FUNCTION_BLOCK FB_LedOff
VAR_INPUT
END_VAR
VAR_OUTPUT
END_VAR
VAR
	state : INT := 0;
	fbSerialSend : FB_SerialCom;
	d0 : BYTE := 16#01;
	d1 : BYTE := 16#44;
	d2 : BYTE := 16#00;
	d3 : BYTE := 16#13;
	d4 : BYTE := 16#00;
	fbSendData : SendData;
END_VAR

(*
BackGroundEL.stOut_EL6002_MB.D[0] := 16#01;
BackGroundEL.stOut_EL6002_MB.D[1] := 16#44;
BackGroundEL.stOut_EL6002_MB.D[2] := 16#00;
BackGroundEL.stOut_EL6002_MB.D[3] := 16#13;
BackGroundEL.stOut_EL6002_MB.D[4] := 16#00;
*)
(*
CASE state OF 
0:
fbSerialSend(
	TxBuffer := GVL.TxBufferEL_MB,
	RxBuffer := GVL.RxBufferEL_MB,
	fbSendData := fbSendData.pSendData,
	Busy =>,
	Error =>
	);
	IF fbSerialSend.Busy = FALSE THEN
		state := state + 1;
	END_IF
1:
fbSerialSend(
	TxBuffer := GVL.TxBufferEL_MB,
	RxBuffer := GVL.RxBufferEL_MB,
	fbSendData := d0,
	Busy =>,
	Error =>
	);
	IF fbSerialSend.Busy = FALSE THEN
		state := state + 1;
	END_IF
2:
fbSerialSend(
	TxBuffer := GVL.TxBufferEL_MB,
	RxBuffer := GVL.RxBufferEL_MB,
	fbSendData := d0,
	Busy =>,
	Error =>
	);
	IF fbSerialSend.Busy = FALSE THEN
		state := state + 1;
	END_IF
3:
fbSerialSend(
	TxBuffer := GVL.TxBufferEL_MB,
	RxBuffer := GVL.RxBufferEL_MB,
	fbSendData := d0,
	Busy =>,
	Error =>
	);
	IF fbSerialSend.Busy = FALSE THEN
		state := state + 1;
	END_IF
4:
fbSerialSend(
	TxBuffer := GVL.TxBufferEL_MB,
	RxBuffer := GVL.RxBufferEL_MB,
	fbSendData := d0,
	Busy =>,
	Error =>
	);
	IF fbSerialSend.Busy = FALSE THEN
		state := 0;
	END_IF
END_CASE
*)

END_FUNCTION_BLOCK

(* stored: Version 1.1.0.1, ProductVersion 3.1.4024.12
   POU FB_LedOff: Id {131b0eb6-a0ec-4892-ad5a-990130f7d082}, SpecialFunc None *)
